{attribute 'enable_dynamic_creation'}
FUNCTION_BLOCK FB_TxtLogger IMPLEMENTS ILogger
VAR_INPUT
END_VAR
VAR_OUTPUT
END_VAR
VAR
END_VAR

METHOD PUBLIC Write : STRING
VAR_INPUT
	sMsg      : STRING;
END_VAR
Write := CONCAT('txt-', sMsg);
// open txt file
// write the message into the txt file
// close txt file
END_METHOD

END_FUNCTION_BLOCK

(* stored: Version 1.1.0.1, ProductVersion 3.1.0.24
   POU FB_TxtLogger: Id {75be9b59-4460-43c6-bf14-70c2bdef8ea6}
   Method Write: Id {eebd0b9d-b1b4-45b5-85bf-6b4d920e6a98} *)
